FUNCTION_BLOCK TestFB EXTENDS StateMachine 
VAR_INPUT
END_VAR
VAR_OUTPUT
	eTestUnitBusyStep : E_TestUnitBusyStep;
END_VAR
VAR
END_VAR

SUPER^();
eTestUnitBusyStep := stStateMachine.uiBusy;
Start();

METHOD PROTECTED Busy : BOOL
stStateMachine.uiBusy := eWAITING_FOR_MATERIAL;
END_METHOD

METHOD PROTECTED Error : BOOL
END_METHOD

METHOD PROTECTED Idle : BOOL
END_METHOD

METHOD PROTECTED Init : BOOL
END_METHOD

METHOD PROTECTED Prepare : BOOL
END_METHOD

METHOD PROTECTED Ready : BOOL
END_METHOD

METHOD PROTECTED Waiting : BOOL
END_METHOD

END_FUNCTION_BLOCK

(* stored: Version 1.1.0.1, ProductVersion 3.1.4024.0
   POU TestFB: Id {67322c55-82fd-4877-8787-835d4a3a6dbc}, SpecialFunc None
   Method Busy: Id {ce67759b-1d29-4132-b761-f69e883f6603}
   Method Error: Id {1d1f7f1a-ccb8-4781-96bb-ad512df84a33}
   Method Idle: Id {694ec343-3079-444c-b1a3-411c4b148a5a}
   Method Init: Id {f578fd0c-2eb8-497d-97cd-787e5f19f5d2}
   Method Prepare: Id {e0e63be2-6199-4de5-b14f-7aa8426fa07f}
   Method Ready: Id {a105b02e-d887-4cc7-83eb-9915747cdccb}
   Method Waiting: Id {46848366-d95a-4684-9298-4f89e58d7989} *)
